FUNCTION_BLOCK SS2_ifb_Base_Fixer (* Template for a Basic Function Block Type *)
  (* Standard: 61499-2 *)
  (* Version 1.0, 2024-07-25, DEVIASH *)
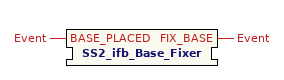
  EVENT_INPUT
    BASE_PLACED; (* Initialization Request *)
  END_EVENT
  EVENT_OUTPUT
    FIX_BASE; (* Initialization Confirm *)
  END_EVENT
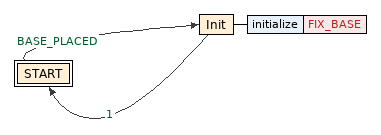
  EC_STATES
    START; (* Initial State *)
    Init : initialize -> FIX_BASE; (* Initialization *)
  END_STATES
  EC_TRANSITIONS
    START TO Init := BASE_PLACED;
    Init TO START := 1;
  END_TRANSITIONS
  ALGORITHM initialize IN ST:

  END_ALGORITHM
END_FUNCTION_BLOCK
